{attribute addProperty BoxType "EL7041-0001-0022"}
{attribute addProperty Id "StatusAT %I*Status_2E2EE8C7162"}
{attribute addProperty CRC "1609782174"}
{attribute addProperty SizeInBites "16"}
{attribute addProperty SizeInBytes "2"}
TYPE STM_Status_5FF3539E :
STRUCT
	{attribute addProperty Name "Status"}
	Status AT %I* : Status_2E2EE8C7;
END_STRUCT
END_TYPE

(* stored: Version 1.2.0.0, ProductVersion 3.1.4024.9
   DUT STM_Status_5FF3539E: Id {a48e14e0-f43c-4590-b4df-31d3cf94f003} *)
